FUNCTION_BLOCK BLINK 
VAR_INPUT
	TimeH: DINT;
	TimeL: DINT;
END_VAR
VAR_OUTPUT
	OUT: BOOL;
END_VAR
VAR
	tonTimeHigh: TON;
	tonTimeLow: TON;
END_VAR

tonTimeLow(IN:= NOT tonTimeHigh.Q , PT:=DINT_TO_TIME(TimeL) , Q=> OUT, ET=> );
tonTimeHigh(IN:=tonTimeLow.Q  , PT:= DINT_TO_TIME(TimeH), Q=> , ET=> );

END_FUNCTION_BLOCK

(* stored: Version 1.1.0.1, ProductVersion 3.1.4022.16
   POU BLINK: Id {2abd3458-a4c2-4604-84be-91318fabc29c}, SpecialFunc None *)
